TEXTLIST ManualText
  0 = ' \n  取料Y轴\n1:初始位 2:Line0取料位 3:Line1取料位 4:Line3取料位\n\n   取料Z轴\n1:上升位 2:下降位_Line0 3:下降位_Line1\n\n   下UC_Y轴\n1:初始位 2:Line2取料位 3:Line3取料位 4:下UC位' | Chinese: ' \n  取料Y轴\n1:初始位 2:Line0取料位 3:Line1取料位 4:Line3取料位\n\n   取料Z轴\n1:上升位 2:下降位_Line0 3:下降位_Line1\n\n   下UC_Y轴\n1:初始位 2:Line2取料位 3:Line3取料位 4:下UC位' | English: ' \nPick the y axis\nThe initial bit is the initial bit 2:line0\n\nPick the z axis\nDrop _line0 3: drop _line1\n\nThe lower uc_y axis\n1: the initial bit 2:line2 takes the material bit \n3:line3 takes the material bit 4: the lower uc bit' | Vietnamese: ' \nL?y v?t li?u trên tr?c Y\n1: ban ??u bit 2: dòng 0 c?p 3: dòng 1 c?p 4: dòng 3 c?p\n\nL?y tr?c Z\n1: n?ng lên 2: h? xu?ng bit _dòng 0 3: h? xu?ng bit _dòng 1\n\nTr?c d??i UC_Y\n1: b?t ??u bit 2: dòng 2 c?p 3: dòng 3 c?p 4: UC'
   = ''
END_TEXTLIST

(* stored: Version 1.1.0.1, ProductVersion 3.1.4024.3
   TextList ManualText: Id {3ad67886-0b61-436a-ac96-59136b45e612} *)
